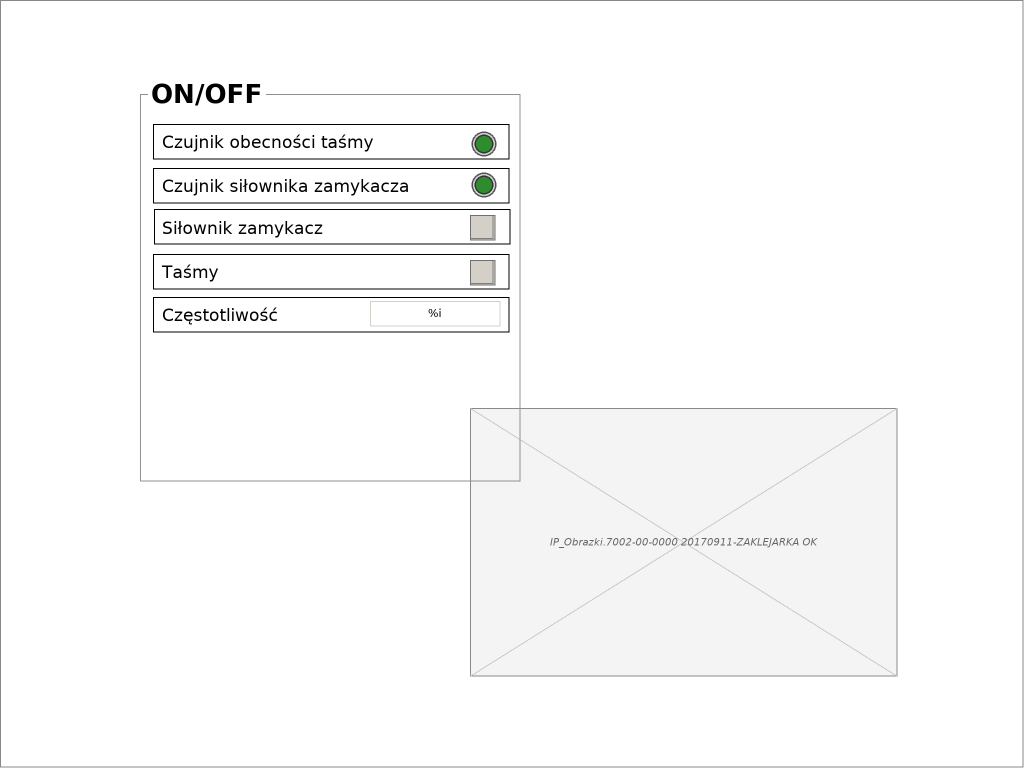
VISUALIZATION Zaklejarka  // 1024x768
    Image (470,408 427x268), image: IP_Obrazki.7002-00-0000 20170911-ZAKLEJARKA OK
    GroupBox (140,86 380x395), "ON/OFF"
        Rectangle (14,123 356x35)
        Rectangle (13,168 356x35)
        Rectangle (13,38 356x35)
        Label (19,41 230x30), "Czujnik obecności taśmy"
        Rectangle (13,82 356x35)
        Label (19,85 239x30), "Czujnik siłownika zamykacza"
        Label (19,171 209x30), "Taśmy"
        Label (19,127 209x30), "Siłownik zamykacz"
        Rectangle (13,211 356x35)
        Lamp1 (330,85 28x28), variable: GVL_Zak_IO.b_kZamykacz1, style: Lamp-Lamp1-Green
        Lamp1 (330,44 28x28), variable: GVL_Zak_IO.b_czujnik_OT, style: Lamp-Lamp1-Green
        Label (19,299 209x30)
        Textfield (230,215 130x25), "%i", text variable: GVL_HMI.iFreqKierownicaMan
            OnMouseClick: write the text variable via Edit
        Button (330,129 25x25), colour toggle: GVL_GLOBAL.zaw_klap_krot_cewka
            tap GVL_HMI.przycisk_sil_zamykacz_zaklejarka
        Button (330,174 25x25), colour toggle: GVL_GLOBAL.tasmy_zaklejarka_cewka
            tap GVL_HMI.przycisk_tasmy_zaklejarka
    Label (159,300 209x30), "Częstotliwość"
END_VISUALIZATION

(* stored: Version 1.1.0.1, ProductVersion 3.1.4022.12
   Visu Zaklejarka: Id {470a3cd3-45c6-4552-b7a3-02598b58f1f4} *)
